(*
used to write all values to and from json files. Will add to lib later
*)

FUNCTION_BLOCK ABSTRACT FB_JsonFile EXTENDS FB_JsonSchemaEx_OLD
VAR_INPUT
END_VAR
VAR_OUTPUT
END_VAR
VAR
END_VAR

END_FUNCTION_BLOCK

(* stored: Version 1.1.0.1, ProductVersion 3.1.4024.12
   POU FB_JsonFile: Id {7d9f6882-413f-46ef-ad72-6dae3775019a}, SpecialFunc None *)
